// TIA Portal V20 export
DATA_BLOCK "Main_Safety_RTG1_DB"   // DB62, F_DB
NAME : FUSI
// stored: InstanceOfName Main_Safety_RTG1, InstanceOfType FB
"Main_Safety_RTG1"
   // VAR
   //    sSupplyPower : Bool;
   //    sAckEmergencyStop : Bool;
   //    sAckFdbPowMach : Bool;
   //    sAckFdbBW_LoaderEstopRelay : Bool;
   //    sAckFdbSonplasDoorClosedRelay : Bool;
   //    ESTOP1_Instance : ESTOP1;
   //    FDBACK_PowerMachine : FDBACK;
   //    FDBACK_BW_LoaderEstopRelay : FDBACK;
   //    FDBACK_SonplasDoorClosedRelay : FDBACK;
   //    DB_ACK_GL : ACK_GL;
   // END_VAR
BEGIN
END_DATA_BLOCK
